FUNCTION CharIsNumberOrMinus : BOOL
VAR_INPUT
	Char : BYTE; // char to check
END_VAR
VAR CONSTANT
	MINUS_ASCII : BYTE := 45;
END_VAR

// check bChar is in numbr range of ascii
CharIsNumberOrMinus := CharIsNumber( Char ) OR_ELSE ( Char = MINUS_ASCII );

END_FUNCTION

(* stored: Version 1.1.0.1, ProductVersion 3.1.4024.0
   POU CharIsNumberOrMinus: Id {3170bf1e-f55e-4533-a163-a665e60a5864}, SpecialFunc None *)
